FUNCTION_BLOCK AX_NOOP (* No-Op, also known as "no Operation" *)
  (* Standard: 61131-3; Classification: standard boolean function; Description: Copyright (c) 2011 TU Wien ACIN, HR Agrartechnik GmbH This program and the accompanying materials are made available under the terms of the Eclipse Public License 2.0 which is available at https://www.eclipse.org/legal/epl-2.0/ SPDX-License-Identifier: EPL-2.0 *)
  (* Version 3.1, 2025-11-04, Franz Höpfinger, HR Agrartechnik GmbH, made AX Version *)
  (* Version 3.0, 2025-04-14, Patrick Aigner, changed package *)
  (* Version 1.0, 2011-06-21, Monika Wenger, TU Wien ACIN *)
  PACKAGE adapter::booleanOperators;
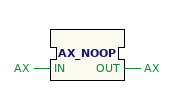
  SOCKETS
    IN : adapter::types::unidirectional::AX; (* Input *)
  END_SOCKETS
  PLUGS
    OUT : adapter::types::unidirectional::AX; (* Output *)
  END_PLUGS
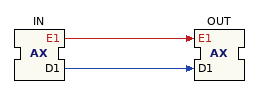
  EVENT_CONNECTIONS
    IN.E1 TO OUT.E1;
  END_CONNECTIONS
  DATA_CONNECTIONS
    IN.D1 TO OUT.D1;
  END_CONNECTIONS
END_FUNCTION_BLOCK
